FUNCTION_BLOCK FB_DigitalOut
VAR_INPUT
	iMaxInCH : INT;
END_VAR
VAR_OUTPUT
END_VAR
VAR

	arDigitalOut 	: ARRAY [1..GVL_DigitalOut.iDoutputChannelCount] OF ST_DigitalOut;
	bLocalDO		: ARRAY [1..GVL_DigitalOut.iDoutputChannelCount] OF BOOL;
	iIndex			: INT;
	iSeqIndex		: INT;
	iMax			: INT;
	arrtrig_output	: ARRAY [1..GVL_DigitalOut.iDoutputChannelCount] OF R_TRIG;
END_VAR
VAR PERSISTENT
	bSafetyDO		: ARRAY [1..GVL_DigitalOut.iDoutputChannelCount] OF BOOL;
END_VAR

AssignDOs();

METHOD AssignDOs : BOOL
VAR_INPUT
END_VAR
VAR
END_VAR
FOR iIndex:=1 TO iMaxInCH BY 1 DO
	GVL_DigitalOut.bDigitalOutFdbk[iIndex] := OutputControl;
END_FOR
END_METHOD

METHOD AssignSafetyChannels : BOOL
VAR_INPUT
END_VAR
bSafetyDO[1]:=TRUE;
bSafetyDO[2]:=TRUE;
bSafetyDO[3]:=TRUE;
bSafetyDO[4]:=TRUE;
END_METHOD

METHOD LimitMaxChannels : BOOL
(*IF iMaxInCH > GVL_DigitalOut.iDoutputChannelCount THEN
	iMax := GVL_DigitalOut.iDoutputChannelCount;
ELSE
	iMax := iMaxInCH;
END_IF
*)

iMax := GVL_DigitalOut.iDoutputChannelCount;
END_METHOD

PROPERTY OutputControl : BOOL
GET
OutputControl:=GVL_DigitalOut.bDigitalOut[iIndex];
END_GET
SET
GVL_DigitalOut.bDigitalOut[iIndex] := OutputControl;
END_SET
END_PROPERTY

END_FUNCTION_BLOCK

(* stored: Version 1.1.0.1, ProductVersion 3.1.4024.12
   POU FB_DigitalOut: Id {aeb990d6-c87d-467f-9591-6e309ab29528}, SpecialFunc None
   Method AssignDOs: Id {5275d904-7606-41ab-9d01-8b3b8085549f}
   Method AssignSafetyChannels: Id {8b5a5991-c603-4533-89bc-314af3e63d29}
   Method LimitMaxChannels: Id {28f1912c-0e14-45c7-9ca2-113bf4b53eae}
   Property OutputControl: Id {2be1f416-be15-4241-a2a6-41167da28aa1}
   Get Get: Id {d4917f0f-8b68-491a-980d-51d3df7226f8}
   Set Set: Id {2e276319-8f76-402f-bad0-1a4cf9260964} *)
